FUNCTION_BLOCK palletOne (* Tamplate for a simple Basic Function Block Type *)
  (* Standard: 61499-2 *)
  (* Version 0.0, 2018-01-05, 4DIAC-IDE, 4DIAC-Consortium *)
  (* Version 1.0, 2016-05-26, AZ, fortiss GmbH *)
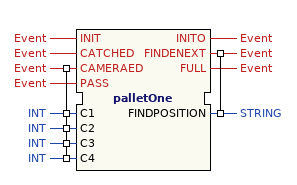
  EVENT_INPUT
    INIT; (* Initialization Request *)
    CATCHED;
    CAMERAED WITH C1, C2, C3, C4;
    PASS;
  END_EVENT
  EVENT_OUTPUT
    INITO; (* Initialization Confirm *)
    FINDENEXT WITH FINDPOSITION; (* Execution Confirmation *)
    FULL;
  END_EVENT
  VAR_INPUT
    C1 : INT; (* Input event qualifier *)
    C2 : INT;
    C3 : INT;
    C4 : INT;
  END_VAR
  VAR_OUTPUT
    FINDPOSITION : STRING;
  END_VAR
  VAR
    pos1 : INT := -1; (* Internal Variable *)
    pos2 : INT := -1; (* Internal Variable *)
    pos3 : INT := -1; (* Internal Variable *)
    pos4 : INT := -1; (* Internal Variable *)
    isFull : BOOL := FALSE; (* Internal Variable *)
    currentPos : INT := 0; (* Internal Variable *)
  END_VAR
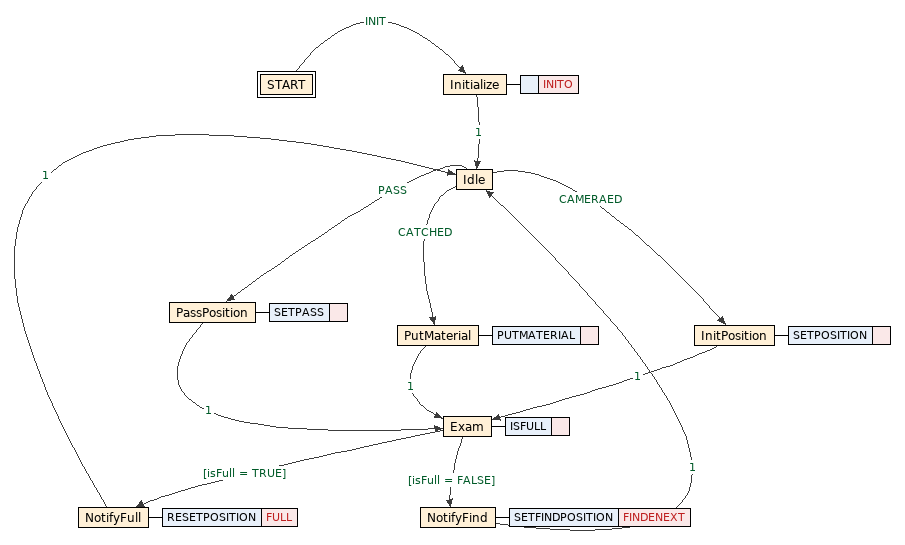
  EC_STATES
    START; (* Initial State *)
    Initialize : -> INITO; (* Initialization *)
    Idle;
    InitPosition : SETPOSITION;
    PutMaterial : PUTMATERIAL;
    NotifyFind : SETFINDPOSITION -> FINDENEXT;
    PassPosition : SETPASS;
    Exam : ISFULL;
    NotifyFull : RESETPOSITION -> FULL;
  END_STATES
  EC_TRANSITIONS
    START TO Initialize := INIT;
    Initialize TO Idle := 1;
    Idle TO InitPosition := CAMERAED;
    Idle TO PutMaterial := CATCHED;
    NotifyFind TO Idle := 1;
    Idle TO PassPosition := PASS;
    PutMaterial TO Exam := 1;
    PassPosition TO Exam := 1;
    Exam TO NotifyFind := [isFull = FALSE];
    Exam TO NotifyFull := [isFull = TRUE];
    NotifyFull TO Idle := 1;
    InitPosition TO Exam := 1;
  END_TRANSITIONS
  ALGORITHM SETPOSITION IN ST: (* new algorithm *)
pos1 := C1;
pos2 := C2;
pos3 := C3;
pos4 := C4;
  END_ALGORITHM
  ALGORITHM PUTMATERIAL IN ST: (* new algorithm *)
IF(currentPos = 1) THEN
	pos1 := 1;
END_IF;

IF(currentPos = 2) THEN
	pos2 := 1;
END_IF;

IF(currentPos = 3) THEN
	pos3 := 1;
END_IF;

IF(currentPos = 4) THEN
	pos4 := 1;
END_IF;
  END_ALGORITHM
  ALGORITHM SETPASS IN ST: (* new algorithm *)
IF(currentPos = 1) THEN
	pos1 := 0;
END_IF;

IF(currentPos = 2) THEN
	pos2 := 0;
END_IF;

IF(currentPos = 3) THEN
	pos3 := 0;
END_IF;

IF(currentPos = 4) THEN
	pos4 := 0;
END_IF
  END_ALGORITHM
  ALGORITHM ISFULL IN ST: (* new algorithm *)
currentPos := 0;
isFull := TRUE;

IF(pos1 = -1) THEN
	currentPos := 1;
	isFull := FALSE;
END_IF;

IF(pos2 = -1) THEN
	currentPos := 2;
	isFull := FALSE;
END_IF;

IF(pos3 = -1) THEN
	currentPos := 3;
	isFull := FALSE;
END_IF;

IF(pos4 = -1) THEN
	currentPos := 4;
	isFull := FALSE;
END_IF;
  END_ALGORITHM
  ALGORITHM RESETPOSITION IN ST: (* new algorithm *)
pos1 := -1;
pos2 := -1;
pos3 := -1;
pos4 := -1;
  END_ALGORITHM
  ALGORITHM SETFINDPOSITION IN ST: (* new algorithm *)
IF(currentPos = 1) THEN
	FINDPOSITION := '22';
END_IF;

IF(currentPos = 2) THEN
	FINDPOSITION := '23';
END_IF;

IF(currentPos = 3) THEN
	FINDPOSITION := '24';
END_IF;

IF(currentPos = 4) THEN
	FINDPOSITION := '26';
END_IF;
  END_ALGORITHM
END_FUNCTION_BLOCK
